FUNCTION_BLOCK F_T_PLC_MS (* reads the internal PLC timer and returns the time *)
  (* Standard: OSCAT; Classification: Measurement *)
  (* Version 0.0, 2011-08-22, 4DIAC-IDE, 4DIAC-Consortium *)
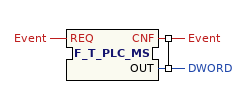
  EVENT_INPUT
    REQ; (* Service Request *)
  END_EVENT
  EVENT_OUTPUT
    CNF WITH OUT; (* Confirmation of Requested Service *)
  END_EVENT
  VAR_OUTPUT
    OUT : DWORD; (* Event Output Qualifier *)
  END_VAR
END_FUNCTION_BLOCK
